FUNCTION_BLOCK ZApp EXTENDS ZApplication.Application
VAR
  _boot : ZAppSequenceBoot;
  _bootFault : ZAppSequenceBootFault;
  _running : ZAppSequenceRunning;
END_VAR

METHOD FB_init : BOOL
VAR_INPUT
  bInitRetains : BOOL; /// if TRUE, the retain variables are initialized (warm start / cold start)
  bInCopyCode : BOOL; /// if TRUE, the instance afterwards gets moved into the copy code (online change)
  displayName : ZCore.ZString;
  com : REFERENCE TO ZApplication.ApplicationComPublish;
END_VAR
SetBootSequence(_boot);
SetBootFaultSequence(_bootFault);
SetRunningSequence(_running);
END_METHOD

END_FUNCTION_BLOCK

(* stored: Version 1.1.0.1
   POU ZApp: Id {bcac29b3-b82e-4456-b732-a1dfcab467d6}, SpecialFunc None
   Method FB_init: Id {b75cf818-75c4-401a-b032-332c8c2e06de} *)
